FUNCTION_BLOCK WAGOConveyorController (* Composite Function Block Type *)
  (* Standard: 61499-2 *)
  (* Version 0.2, 2003-12-05, JHC, Rockwell Automation, Renamed from NEWCOMPFB. *)
  (* Compiler header: package fb.rt.wago; *)
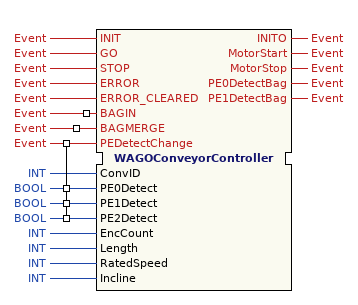
  EVENT_INPUT
    INIT; (* Initialization Request *)
    GO; (* Normal Execution Request *)
    STOP; (* Normal Execution Request *)
    ERROR; (* Normal Execution Request *)
    ERROR_CLEARED; (* Normal Execution Request *)
    BAGIN WITH BagDataIn;
    BAGMERGE WITH BagMergeIn;
    PEDetectChange WITH PE0Detect, PE1Detect, PE2Detect; (* Instance of Time *)
  END_EVENT
  EVENT_OUTPUT
    INITO; (* Initialization Confirm *)
    MotorStart;
    MotorStop;
    PE0DetectBag;
    PE1DetectBag;
  END_EVENT
  VAR_INPUT
    ConvID : INT; (* Input event qualifier *)
    PE0Detect : BOOL; (* Input event qualifier *)
    PE1Detect : BOOL; (* Input event qualifier *)
    PE2Detect : BOOL; (* Input event qualifier *)
    EncCount : INT;
    Length : INT;
    RatedSpeed : INT;
    Incline : INT;
  END_VAR
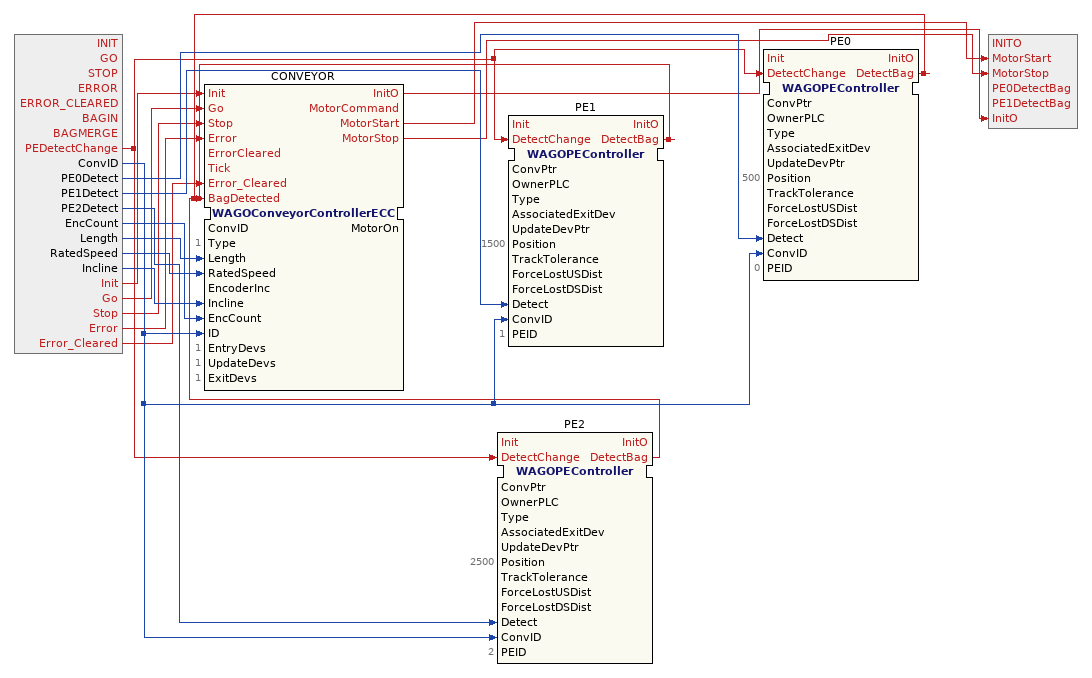
  FBS
    CONVEYOR : WAGOConveyorControllerECC(Type := 1, EntryDevs := 1, UpdateDevs := 1, ExitDevs := 1);
    PE0 : WAGOPEController(PEID := 0, Position := 500);
    PE1 : WAGOPEController(PEID := 1, Position := 1500);
    PE2 : WAGOPEController(PEID := 2, Position := 2500);
  END_FBS
  EVENT_CONNECTIONS
    Init TO CONVEYOR.Init;
    CONVEYOR.InitO TO InitO;
    Go TO CONVEYOR.Go;
    Stop TO CONVEYOR.Stop;
    Error TO CONVEYOR.Error;
    Error_Cleared TO CONVEYOR.Error_Cleared;
    CONVEYOR.MotorStart TO MotorStart;
    CONVEYOR.MotorStop TO MotorStop;
    PE0.DetectBag TO CONVEYOR.BagDetected;
    PE1.DetectBag TO CONVEYOR.BagDetected;
    PE2.DetectBag TO CONVEYOR.BagDetected;
    PEDetectChange TO PE0.DetectChange;
    PEDetectChange TO PE1.DetectChange;
    PEDetectChange TO PE2.DetectChange;
  END_CONNECTIONS
  DATA_CONNECTIONS
    EncCount TO CONVEYOR.EncCount;
    Length TO CONVEYOR.Length;
    RatedSpeed TO CONVEYOR.RatedSpeed;
    Incline TO CONVEYOR.Incline;
    ConvID TO CONVEYOR.ID;
    ConvID TO PE0.ConvID;
    ConvID TO PE1.ConvID;
    ConvID TO PE2.ConvID;
    PE0Detect TO PE0.Detect;
    PE1Detect TO PE1.Detect;
    PE2Detect TO PE2.Detect;
  END_CONNECTIONS
END_FUNCTION_BLOCK
